TYPE DUT_SENSOR_DATAS_4 :
UNION
	data_lreal:REAL;
	data_byte:ARRAY[0..3] OF BYTE;
END_UNION
END_TYPE

(* stored: Version 1.1.0.1, ProductVersion 3.1.4024.6
   DUT DUT_SENSOR_DATAS_4: Id {6e6638b4-028e-40f2-851f-43ed7d1b36ec} *)
